// TIA Portal V19 export
DATA_BLOCK "MonitoringValves_DB"   // DB21
VERSION : 0.0
// stored: AutoNumber false, InstanceOfName MonitoringValves, InstanceOfType FB
"MonitoringValves"
   // VAR
   //    V01_01 : "ValveMonitor";
   //    V01_03 : "ValveMonitor";
   //    V01_04 : "ValveMonitor";
   //    V01_08 : "ValveMonitor";
   //    V01_09 : "ValveMonitor";
   //    V01_11 : "ValveMonitor";
   //    V01_12 : "ValveMonitor";
   //    V01_13 : "ValveMonitor";
   //    V01_14 : "ValveMonitor";
   //    V01_15 : "ValveMonitor";
   //    V01_16 : "ValveMonitor";
   //    V01_17 : "ValveMonitor";
   //    V09_01 : "ValveMonitor";
   //    V09_02 : "ValveMonitor";
   //    V09_03 : "ValveMonitor";
   //    V09_04 : "ValveMonitor";
   //    V09_05 : "ValveMonitor";
   //    V09_06 : "ValveMonitor";
   //    V09_07 : "ValveMonitor";
   //    V09_08 : "ValveMonitor";
   //    V09_09 : "ValveMonitor";
   //    V09_10 : "ValveMonitor";
   //    V09_11 : "ValveMonitor";
   //    V09_12 : "ValveMonitor";
   // END_VAR
BEGIN
END_DATA_BLOCK
